(* CoDeSys 2.3.9.62 project: Tema2Ejemplo2-Sol1-Deposito.pro *)

(* Global variable list: Global_Variables *)
VAR_GLOBAL
  A:BOOL;
  B:BOOL;
  Bomba:BOOL;
  Bomba1:BOOL;
	Encendido:BOOL;
END_VAR

(* POU PLC_PRG, ST *)
PROGRAM PLC_PRG
VAR
  posy:INT;

	Desague: BOOL;
END_VAR
Control();


IF Bomba=TRUE THEN
IF posy>-187 THEN
  posy:=posy-1;
END_IF
END_IF

IF Bomba=FALSE THEN
IF posy<52 THEN
  posy:=posy+1;
END_IF
END_IF

IF Bomba1=TRUE THEN
IF posy>-187 THEN
  posy:=posy-1;
END_IF
END_IF


IF Desague=1 THEN
IF posy<48 THEN
posy:=posy+4;
END_IF
END_IF

IF posy<-121 THEN
  A:=TRUE;
ELSE
  A:=FALSE;
END_IF

IF posy<-166 THEN
  B:=TRUE;
ELSE
  B:=FALSE;
END_IF
END_PROGRAM

(* POU Control, LD *)
PROGRAM Control
VAR
 X:BOOL;
END_VAR
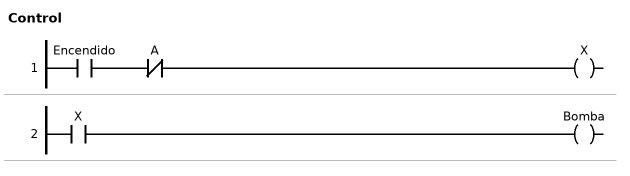
_LD_ (* Ladder Diagram *)
NETWORK 1
	[Encendido] - [/A] --- (X)
NETWORK 2
	[X] --- (Bomba)
_END_LD_
(* the same logic as Structured Text *)
(* Network 1 *)
X := Encendido AND NOT A;
(* Network 2 *)
Bomba := X;
END_PROGRAM

(* Visualisation Deposito
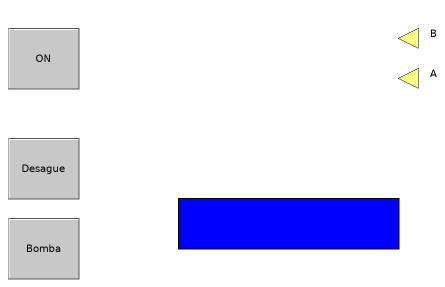
button at (50,80)-(121,141): text "ON"; toggles .Encendido
button at (50,190)-(121,251): text "Desague"; toggles PLC_PRG.Desague
polygon at (440,80)-(460,100): alarm colour if .B; toggles .B
polygon at (440,120)-(460,140): alarm colour if .A; toggles .A
button at (50,270)-(121,331): text "Bomba"; toggles .Bomba1
rectangle at (460,70)-(491,101): text "B"
rectangle at (460,110)-(491,141): text "A"
rectangle at (220,250)-(441,301): top PLC_PRG.posy
1 more shapes without text or variables
1 elements of other kinds (tables, trends, ...) not read
*)
